// TIA Portal V20 export
FUNCTION "SafetyDoor" : Void   // FC97, LAD
// stored: SetENOAutomatically false
   VAR CONSTANT
      TRUE : Bool := TRUE;
      FALSE : Bool;
   END_VAR
   VAR_TEMP   // added for the SCL form of the ladder/FBD networks
      _w1 : Bool;
   END_VAR
BEGIN

REGION Network 1: fDoor1 monitoring
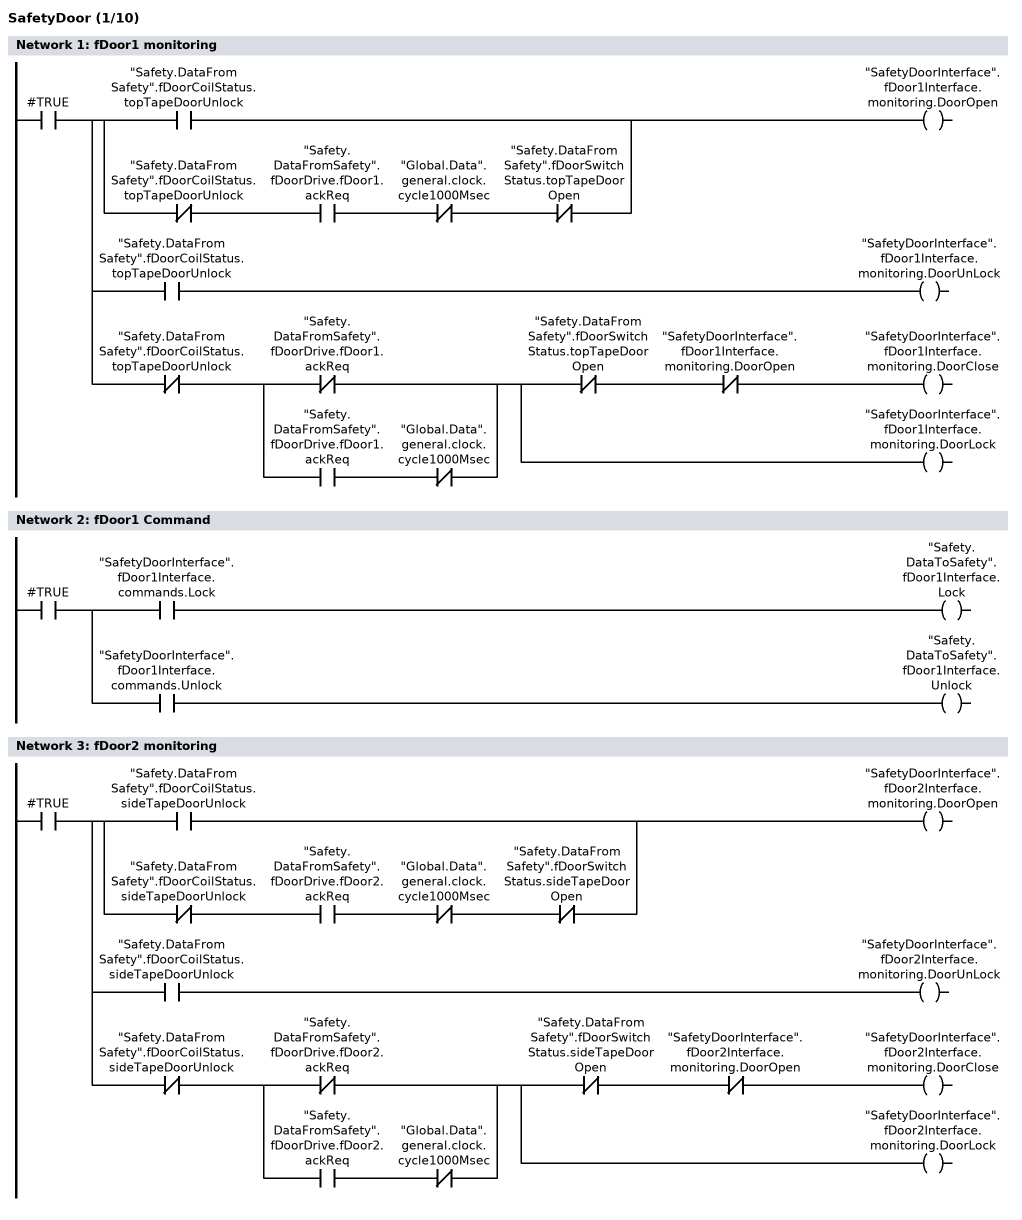
   RUNG wire#powerrail
      Contact( #TRUE )
      wire#w1
      Contact( "Safety.DataFromSafety".fDoorCoilStatus.topTapeDoorUnlock )
      wire#w2
      Coil( "SafetyDoorInterface".fDoor1Interface.monitoring.DoorOpen )
   END_RUNG
   RUNG wire#w1
      I_Contact( "Safety.DataFromSafety".fDoorCoilStatus.topTapeDoorUnlock )
      Contact( "Safety.DataFromSafety".fDoorDrive.fDoor1.ackReq )
      I_Contact( "Global.Data".general.clock.cycle1000Msec )
      I_Contact( "Safety.DataFromSafety".fDoorSwitchStatus.topTapeDoorOpen )
   END_RUNG wire#w2
   RUNG wire#w1
      Contact( "Safety.DataFromSafety".fDoorCoilStatus.topTapeDoorUnlock )
      Coil( "SafetyDoorInterface".fDoor1Interface.monitoring.DoorUnLock )
   END_RUNG
   RUNG wire#w1
      I_Contact( "Safety.DataFromSafety".fDoorCoilStatus.topTapeDoorUnlock )
      wire#w3
      I_Contact( "Safety.DataFromSafety".fDoorDrive.fDoor1.ackReq )
      wire#w4
      I_Contact( "Safety.DataFromSafety".fDoorSwitchStatus.topTapeDoorOpen )
      I_Contact( "SafetyDoorInterface".fDoor1Interface.monitoring.DoorOpen )
      Coil( "SafetyDoorInterface".fDoor1Interface.monitoring.DoorClose )
   END_RUNG
   RUNG wire#w3
      Contact( "Safety.DataFromSafety".fDoorDrive.fDoor1.ackReq )
      I_Contact( "Global.Data".general.clock.cycle1000Msec )
   END_RUNG wire#w4
   RUNG wire#w4
      Coil( "SafetyDoorInterface".fDoor1Interface.monitoring.DoorLock )
   END_RUNG
   // the same network as SCL:
   "SafetyDoorInterface".fDoor1Interface.monitoring.DoorOpen := #TRUE AND ("Safety.DataFromSafety".fDoorCoilStatus.topTapeDoorUnlock OR (NOT "Safety.DataFromSafety".fDoorCoilStatus.topTapeDoorUnlock AND "Safety.DataFromSafety".fDoorDrive.fDoor1.ackReq AND NOT "Global.Data".general.clock.cycle1000Msec AND NOT "Safety.DataFromSafety".fDoorSwitchStatus.topTapeDoorOpen));
   "SafetyDoorInterface".fDoor1Interface.monitoring.DoorUnLock := #TRUE AND "Safety.DataFromSafety".fDoorCoilStatus.topTapeDoorUnlock;
   #_w1 := #TRUE AND NOT "Safety.DataFromSafety".fDoorCoilStatus.topTapeDoorUnlock AND (NOT "Safety.DataFromSafety".fDoorDrive.fDoor1.ackReq OR ("Safety.DataFromSafety".fDoorDrive.fDoor1.ackReq AND NOT "Global.Data".general.clock.cycle1000Msec));
   "SafetyDoorInterface".fDoor1Interface.monitoring.DoorClose := #_w1 AND NOT "Safety.DataFromSafety".fDoorSwitchStatus.topTapeDoorOpen AND NOT "SafetyDoorInterface".fDoor1Interface.monitoring.DoorOpen;
   "SafetyDoorInterface".fDoor1Interface.monitoring.DoorLock := #_w1;
END_REGION

REGION Network 2: fDoor1 Command
   RUNG wire#powerrail
      Contact( #TRUE )
      wire#w1
      Contact( "SafetyDoorInterface".fDoor1Interface.commands.Lock )
      Coil( "Safety.DataToSafety".fDoor1Interface.Lock )
   END_RUNG
   RUNG wire#w1
      Contact( "SafetyDoorInterface".fDoor1Interface.commands.Unlock )
      Coil( "Safety.DataToSafety".fDoor1Interface.Unlock )
   END_RUNG
   // the same network as SCL:
   "Safety.DataToSafety".fDoor1Interface.Lock := #TRUE AND "SafetyDoorInterface".fDoor1Interface.commands.Lock;
   "Safety.DataToSafety".fDoor1Interface.Unlock := #TRUE AND "SafetyDoorInterface".fDoor1Interface.commands.Unlock;
END_REGION

REGION Network 3: fDoor2 monitoring
   RUNG wire#powerrail
      Contact( #TRUE )
      wire#w1
      Contact( "Safety.DataFromSafety".fDoorCoilStatus.sideTapeDoorUnlock )
      wire#w2
      Coil( "SafetyDoorInterface".fDoor2Interface.monitoring.DoorOpen )
   END_RUNG
   RUNG wire#w1
      I_Contact( "Safety.DataFromSafety".fDoorCoilStatus.sideTapeDoorUnlock )
      Contact( "Safety.DataFromSafety".fDoorDrive.fDoor2.ackReq )
      I_Contact( "Global.Data".general.clock.cycle1000Msec )
      I_Contact( "Safety.DataFromSafety".fDoorSwitchStatus.sideTapeDoorOpen )
   END_RUNG wire#w2
   RUNG wire#w1
      Contact( "Safety.DataFromSafety".fDoorCoilStatus.sideTapeDoorUnlock )
      Coil( "SafetyDoorInterface".fDoor2Interface.monitoring.DoorUnLock )
   END_RUNG
   RUNG wire#w1
      I_Contact( "Safety.DataFromSafety".fDoorCoilStatus.sideTapeDoorUnlock )
      wire#w3
      I_Contact( "Safety.DataFromSafety".fDoorDrive.fDoor2.ackReq )
      wire#w4
      I_Contact( "Safety.DataFromSafety".fDoorSwitchStatus.sideTapeDoorOpen )
      I_Contact( "SafetyDoorInterface".fDoor2Interface.monitoring.DoorOpen )
      Coil( "SafetyDoorInterface".fDoor2Interface.monitoring.DoorClose )
   END_RUNG
   RUNG wire#w3
      Contact( "Safety.DataFromSafety".fDoorDrive.fDoor2.ackReq )
      I_Contact( "Global.Data".general.clock.cycle1000Msec )
   END_RUNG wire#w4
   RUNG wire#w4
      Coil( "SafetyDoorInterface".fDoor2Interface.monitoring.DoorLock )
   END_RUNG
   // the same network as SCL:
   "SafetyDoorInterface".fDoor2Interface.monitoring.DoorOpen := #TRUE AND ("Safety.DataFromSafety".fDoorCoilStatus.sideTapeDoorUnlock OR (NOT "Safety.DataFromSafety".fDoorCoilStatus.sideTapeDoorUnlock AND "Safety.DataFromSafety".fDoorDrive.fDoor2.ackReq AND NOT "Global.Data".general.clock.cycle1000Msec AND NOT "Safety.DataFromSafety".fDoorSwitchStatus.sideTapeDoorOpen));
   "SafetyDoorInterface".fDoor2Interface.monitoring.DoorUnLock := #TRUE AND "Safety.DataFromSafety".fDoorCoilStatus.sideTapeDoorUnlock;
   #_w1 := #TRUE AND NOT "Safety.DataFromSafety".fDoorCoilStatus.sideTapeDoorUnlock AND (NOT "Safety.DataFromSafety".fDoorDrive.fDoor2.ackReq OR ("Safety.DataFromSafety".fDoorDrive.fDoor2.ackReq AND NOT "Global.Data".general.clock.cycle1000Msec));
   "SafetyDoorInterface".fDoor2Interface.monitoring.DoorClose := #_w1 AND NOT "Safety.DataFromSafety".fDoorSwitchStatus.sideTapeDoorOpen AND NOT "SafetyDoorInterface".fDoor2Interface.monitoring.DoorOpen;
   "SafetyDoorInterface".fDoor2Interface.monitoring.DoorLock := #_w1;
END_REGION

REGION Network 4: fDoor2 Command
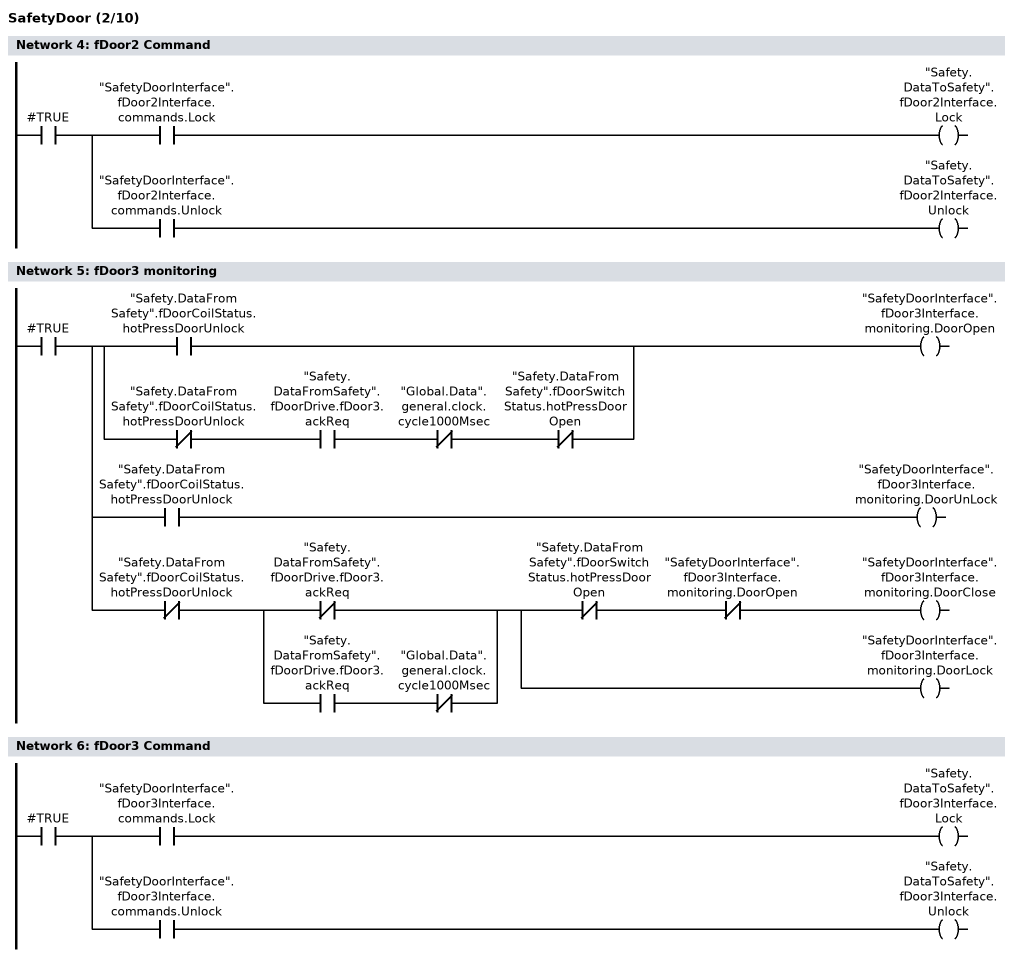
   RUNG wire#powerrail
      Contact( #TRUE )
      wire#w1
      Contact( "SafetyDoorInterface".fDoor2Interface.commands.Lock )
      Coil( "Safety.DataToSafety".fDoor2Interface.Lock )
   END_RUNG
   RUNG wire#w1
      Contact( "SafetyDoorInterface".fDoor2Interface.commands.Unlock )
      Coil( "Safety.DataToSafety".fDoor2Interface.Unlock )
   END_RUNG
   // the same network as SCL:
   "Safety.DataToSafety".fDoor2Interface.Lock := #TRUE AND "SafetyDoorInterface".fDoor2Interface.commands.Lock;
   "Safety.DataToSafety".fDoor2Interface.Unlock := #TRUE AND "SafetyDoorInterface".fDoor2Interface.commands.Unlock;
END_REGION

REGION Network 5: fDoor3 monitoring
   RUNG wire#powerrail
      Contact( #TRUE )
      wire#w1
      Contact( "Safety.DataFromSafety".fDoorCoilStatus.hotPressDoorUnlock )
      wire#w2
      Coil( "SafetyDoorInterface".fDoor3Interface.monitoring.DoorOpen )
   END_RUNG
   RUNG wire#w1
      I_Contact( "Safety.DataFromSafety".fDoorCoilStatus.hotPressDoorUnlock )
      Contact( "Safety.DataFromSafety".fDoorDrive.fDoor3.ackReq )
      I_Contact( "Global.Data".general.clock.cycle1000Msec )
      I_Contact( "Safety.DataFromSafety".fDoorSwitchStatus.hotPressDoorOpen )
   END_RUNG wire#w2
   RUNG wire#w1
      Contact( "Safety.DataFromSafety".fDoorCoilStatus.hotPressDoorUnlock )
      Coil( "SafetyDoorInterface".fDoor3Interface.monitoring.DoorUnLock )
   END_RUNG
   RUNG wire#w1
      I_Contact( "Safety.DataFromSafety".fDoorCoilStatus.hotPressDoorUnlock )
      wire#w3
      I_Contact( "Safety.DataFromSafety".fDoorDrive.fDoor3.ackReq )
      wire#w4
      I_Contact( "Safety.DataFromSafety".fDoorSwitchStatus.hotPressDoorOpen )
      I_Contact( "SafetyDoorInterface".fDoor3Interface.monitoring.DoorOpen )
      Coil( "SafetyDoorInterface".fDoor3Interface.monitoring.DoorClose )
   END_RUNG
   RUNG wire#w3
      Contact( "Safety.DataFromSafety".fDoorDrive.fDoor3.ackReq )
      I_Contact( "Global.Data".general.clock.cycle1000Msec )
   END_RUNG wire#w4
   RUNG wire#w4
      Coil( "SafetyDoorInterface".fDoor3Interface.monitoring.DoorLock )
   END_RUNG
   // the same network as SCL:
   "SafetyDoorInterface".fDoor3Interface.monitoring.DoorOpen := #TRUE AND ("Safety.DataFromSafety".fDoorCoilStatus.hotPressDoorUnlock OR (NOT "Safety.DataFromSafety".fDoorCoilStatus.hotPressDoorUnlock AND "Safety.DataFromSafety".fDoorDrive.fDoor3.ackReq AND NOT "Global.Data".general.clock.cycle1000Msec AND NOT "Safety.DataFromSafety".fDoorSwitchStatus.hotPressDoorOpen));
   "SafetyDoorInterface".fDoor3Interface.monitoring.DoorUnLock := #TRUE AND "Safety.DataFromSafety".fDoorCoilStatus.hotPressDoorUnlock;
   #_w1 := #TRUE AND NOT "Safety.DataFromSafety".fDoorCoilStatus.hotPressDoorUnlock AND (NOT "Safety.DataFromSafety".fDoorDrive.fDoor3.ackReq OR ("Safety.DataFromSafety".fDoorDrive.fDoor3.ackReq AND NOT "Global.Data".general.clock.cycle1000Msec));
   "SafetyDoorInterface".fDoor3Interface.monitoring.DoorClose := #_w1 AND NOT "Safety.DataFromSafety".fDoorSwitchStatus.hotPressDoorOpen AND NOT "SafetyDoorInterface".fDoor3Interface.monitoring.DoorOpen;
   "SafetyDoorInterface".fDoor3Interface.monitoring.DoorLock := #_w1;
END_REGION

REGION Network 6: fDoor3 Command
   RUNG wire#powerrail
      Contact( #TRUE )
      wire#w1
      Contact( "SafetyDoorInterface".fDoor3Interface.commands.Lock )
      Coil( "Safety.DataToSafety".fDoor3Interface.Lock )
   END_RUNG
   RUNG wire#w1
      Contact( "SafetyDoorInterface".fDoor3Interface.commands.Unlock )
      Coil( "Safety.DataToSafety".fDoor3Interface.Unlock )
   END_RUNG
   // the same network as SCL:
   "Safety.DataToSafety".fDoor3Interface.Lock := #TRUE AND "SafetyDoorInterface".fDoor3Interface.commands.Lock;
   "Safety.DataToSafety".fDoor3Interface.Unlock := #TRUE AND "SafetyDoorInterface".fDoor3Interface.commands.Unlock;
END_REGION

REGION Network 7: fDoor4 monitoring
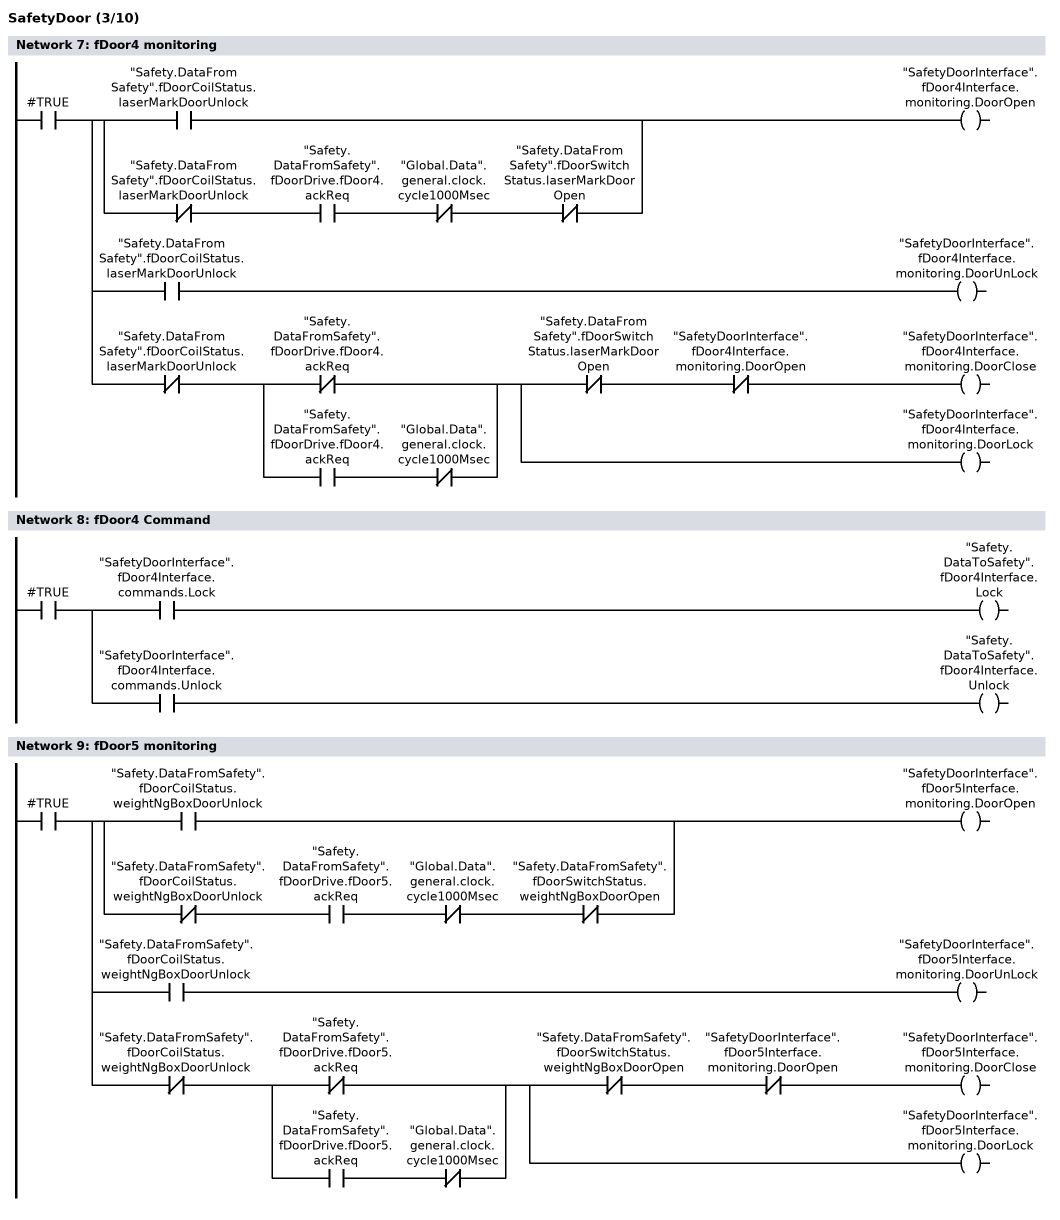
   RUNG wire#powerrail
      Contact( #TRUE )
      wire#w1
      Contact( "Safety.DataFromSafety".fDoorCoilStatus.laserMarkDoorUnlock )
      wire#w2
      Coil( "SafetyDoorInterface".fDoor4Interface.monitoring.DoorOpen )
   END_RUNG
   RUNG wire#w1
      I_Contact( "Safety.DataFromSafety".fDoorCoilStatus.laserMarkDoorUnlock )
      Contact( "Safety.DataFromSafety".fDoorDrive.fDoor4.ackReq )
      I_Contact( "Global.Data".general.clock.cycle1000Msec )
      I_Contact( "Safety.DataFromSafety".fDoorSwitchStatus.laserMarkDoorOpen )
   END_RUNG wire#w2
   RUNG wire#w1
      Contact( "Safety.DataFromSafety".fDoorCoilStatus.laserMarkDoorUnlock )
      Coil( "SafetyDoorInterface".fDoor4Interface.monitoring.DoorUnLock )
   END_RUNG
   RUNG wire#w1
      I_Contact( "Safety.DataFromSafety".fDoorCoilStatus.laserMarkDoorUnlock )
      wire#w3
      I_Contact( "Safety.DataFromSafety".fDoorDrive.fDoor4.ackReq )
      wire#w4
      I_Contact( "Safety.DataFromSafety".fDoorSwitchStatus.laserMarkDoorOpen )
      I_Contact( "SafetyDoorInterface".fDoor4Interface.monitoring.DoorOpen )
      Coil( "SafetyDoorInterface".fDoor4Interface.monitoring.DoorClose )
   END_RUNG
   RUNG wire#w3
      Contact( "Safety.DataFromSafety".fDoorDrive.fDoor4.ackReq )
      I_Contact( "Global.Data".general.clock.cycle1000Msec )
   END_RUNG wire#w4
   RUNG wire#w4
      Coil( "SafetyDoorInterface".fDoor4Interface.monitoring.DoorLock )
   END_RUNG
   // the same network as SCL:
   "SafetyDoorInterface".fDoor4Interface.monitoring.DoorOpen := #TRUE AND ("Safety.DataFromSafety".fDoorCoilStatus.laserMarkDoorUnlock OR (NOT "Safety.DataFromSafety".fDoorCoilStatus.laserMarkDoorUnlock AND "Safety.DataFromSafety".fDoorDrive.fDoor4.ackReq AND NOT "Global.Data".general.clock.cycle1000Msec AND NOT "Safety.DataFromSafety".fDoorSwitchStatus.laserMarkDoorOpen));
   "SafetyDoorInterface".fDoor4Interface.monitoring.DoorUnLock := #TRUE AND "Safety.DataFromSafety".fDoorCoilStatus.laserMarkDoorUnlock;
   #_w1 := #TRUE AND NOT "Safety.DataFromSafety".fDoorCoilStatus.laserMarkDoorUnlock AND (NOT "Safety.DataFromSafety".fDoorDrive.fDoor4.ackReq OR ("Safety.DataFromSafety".fDoorDrive.fDoor4.ackReq AND NOT "Global.Data".general.clock.cycle1000Msec));
   "SafetyDoorInterface".fDoor4Interface.monitoring.DoorClose := #_w1 AND NOT "Safety.DataFromSafety".fDoorSwitchStatus.laserMarkDoorOpen AND NOT "SafetyDoorInterface".fDoor4Interface.monitoring.DoorOpen;
   "SafetyDoorInterface".fDoor4Interface.monitoring.DoorLock := #_w1;
END_REGION

REGION Network 8: fDoor4 Command
   RUNG wire#powerrail
      Contact( #TRUE )
      wire#w1
      Contact( "SafetyDoorInterface".fDoor4Interface.commands.Lock )
      Coil( "Safety.DataToSafety".fDoor4Interface.Lock )
   END_RUNG
   RUNG wire#w1
      Contact( "SafetyDoorInterface".fDoor4Interface.commands.Unlock )
      Coil( "Safety.DataToSafety".fDoor4Interface.Unlock )
   END_RUNG
   // the same network as SCL:
   "Safety.DataToSafety".fDoor4Interface.Lock := #TRUE AND "SafetyDoorInterface".fDoor4Interface.commands.Lock;
   "Safety.DataToSafety".fDoor4Interface.Unlock := #TRUE AND "SafetyDoorInterface".fDoor4Interface.commands.Unlock;
END_REGION

REGION Network 9: fDoor5 monitoring
   RUNG wire#powerrail
      Contact( #TRUE )
      wire#w1
      Contact( "Safety.DataFromSafety".fDoorCoilStatus.weightNgBoxDoorUnlock )
      wire#w2
      Coil( "SafetyDoorInterface".fDoor5Interface.monitoring.DoorOpen )
   END_RUNG
   RUNG wire#w1
      I_Contact( "Safety.DataFromSafety".fDoorCoilStatus.weightNgBoxDoorUnlock )
      Contact( "Safety.DataFromSafety".fDoorDrive.fDoor5.ackReq )
      I_Contact( "Global.Data".general.clock.cycle1000Msec )
      I_Contact( "Safety.DataFromSafety".fDoorSwitchStatus.weightNgBoxDoorOpen )
   END_RUNG wire#w2
   RUNG wire#w1
      Contact( "Safety.DataFromSafety".fDoorCoilStatus.weightNgBoxDoorUnlock )
      Coil( "SafetyDoorInterface".fDoor5Interface.monitoring.DoorUnLock )
   END_RUNG
   RUNG wire#w1
      I_Contact( "Safety.DataFromSafety".fDoorCoilStatus.weightNgBoxDoorUnlock )
      wire#w3
      I_Contact( "Safety.DataFromSafety".fDoorDrive.fDoor5.ackReq )
      wire#w4
      I_Contact( "Safety.DataFromSafety".fDoorSwitchStatus.weightNgBoxDoorOpen )
      I_Contact( "SafetyDoorInterface".fDoor5Interface.monitoring.DoorOpen )
      Coil( "SafetyDoorInterface".fDoor5Interface.monitoring.DoorClose )
   END_RUNG
   RUNG wire#w3
      Contact( "Safety.DataFromSafety".fDoorDrive.fDoor5.ackReq )
      I_Contact( "Global.Data".general.clock.cycle1000Msec )
   END_RUNG wire#w4
   RUNG wire#w4
      Coil( "SafetyDoorInterface".fDoor5Interface.monitoring.DoorLock )
   END_RUNG
   // the same network as SCL:
   "SafetyDoorInterface".fDoor5Interface.monitoring.DoorOpen := #TRUE AND ("Safety.DataFromSafety".fDoorCoilStatus.weightNgBoxDoorUnlock OR (NOT "Safety.DataFromSafety".fDoorCoilStatus.weightNgBoxDoorUnlock AND "Safety.DataFromSafety".fDoorDrive.fDoor5.ackReq AND NOT "Global.Data".general.clock.cycle1000Msec AND NOT "Safety.DataFromSafety".fDoorSwitchStatus.weightNgBoxDoorOpen));
   "SafetyDoorInterface".fDoor5Interface.monitoring.DoorUnLock := #TRUE AND "Safety.DataFromSafety".fDoorCoilStatus.weightNgBoxDoorUnlock;
   #_w1 := #TRUE AND NOT "Safety.DataFromSafety".fDoorCoilStatus.weightNgBoxDoorUnlock AND (NOT "Safety.DataFromSafety".fDoorDrive.fDoor5.ackReq OR ("Safety.DataFromSafety".fDoorDrive.fDoor5.ackReq AND NOT "Global.Data".general.clock.cycle1000Msec));
   "SafetyDoorInterface".fDoor5Interface.monitoring.DoorClose := #_w1 AND NOT "Safety.DataFromSafety".fDoorSwitchStatus.weightNgBoxDoorOpen AND NOT "SafetyDoorInterface".fDoor5Interface.monitoring.DoorOpen;
   "SafetyDoorInterface".fDoor5Interface.monitoring.DoorLock := #_w1;
END_REGION

REGION Network 10: fDoor5 Command
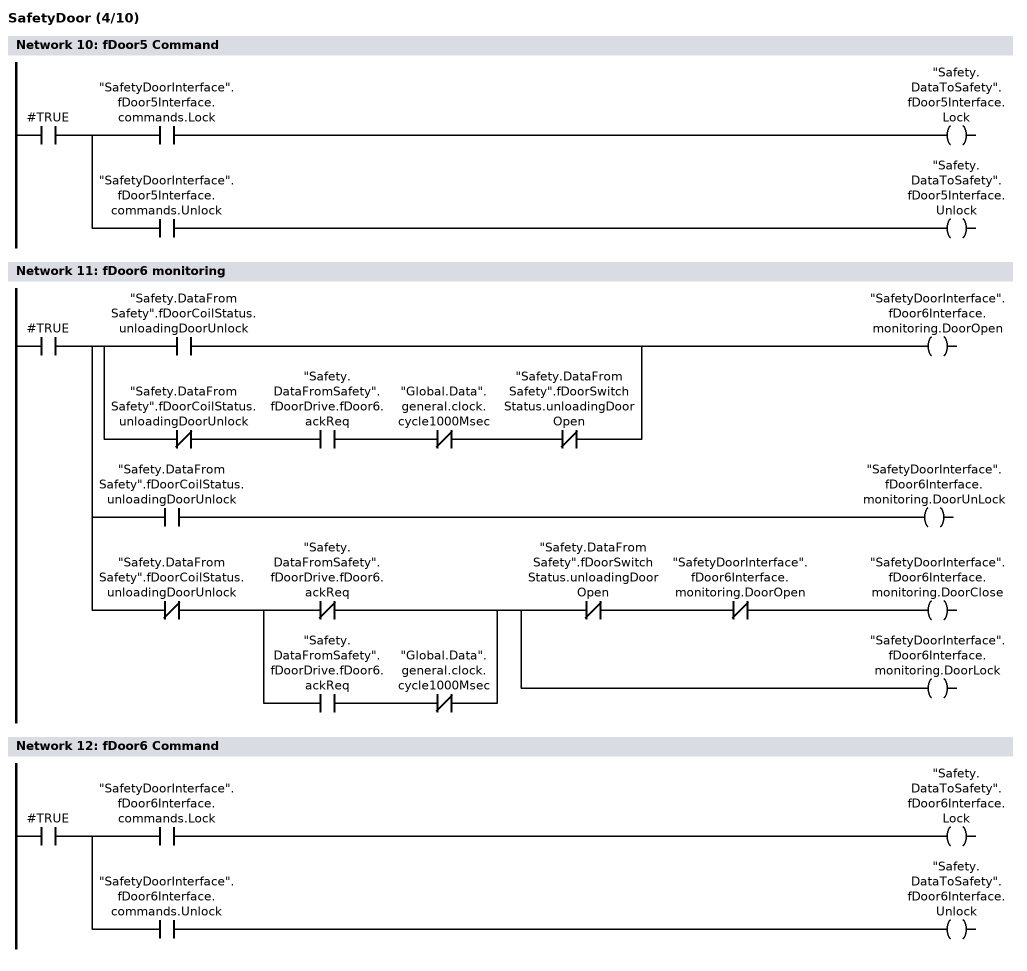
   RUNG wire#powerrail
      Contact( #TRUE )
      wire#w1
      Contact( "SafetyDoorInterface".fDoor5Interface.commands.Lock )
      Coil( "Safety.DataToSafety".fDoor5Interface.Lock )
   END_RUNG
   RUNG wire#w1
      Contact( "SafetyDoorInterface".fDoor5Interface.commands.Unlock )
      Coil( "Safety.DataToSafety".fDoor5Interface.Unlock )
   END_RUNG
   // the same network as SCL:
   "Safety.DataToSafety".fDoor5Interface.Lock := #TRUE AND "SafetyDoorInterface".fDoor5Interface.commands.Lock;
   "Safety.DataToSafety".fDoor5Interface.Unlock := #TRUE AND "SafetyDoorInterface".fDoor5Interface.commands.Unlock;
END_REGION

REGION Network 11: fDoor6 monitoring
   RUNG wire#powerrail
      Contact( #TRUE )
      wire#w1
      Contact( "Safety.DataFromSafety".fDoorCoilStatus.unloadingDoorUnlock )
      wire#w2
      Coil( "SafetyDoorInterface".fDoor6Interface.monitoring.DoorOpen )
   END_RUNG
   RUNG wire#w1
      I_Contact( "Safety.DataFromSafety".fDoorCoilStatus.unloadingDoorUnlock )
      Contact( "Safety.DataFromSafety".fDoorDrive.fDoor6.ackReq )
      I_Contact( "Global.Data".general.clock.cycle1000Msec )
      I_Contact( "Safety.DataFromSafety".fDoorSwitchStatus.unloadingDoorOpen )
   END_RUNG wire#w2
   RUNG wire#w1
      Contact( "Safety.DataFromSafety".fDoorCoilStatus.unloadingDoorUnlock )
      Coil( "SafetyDoorInterface".fDoor6Interface.monitoring.DoorUnLock )
   END_RUNG
   RUNG wire#w1
      I_Contact( "Safety.DataFromSafety".fDoorCoilStatus.unloadingDoorUnlock )
      wire#w3
      I_Contact( "Safety.DataFromSafety".fDoorDrive.fDoor6.ackReq )
      wire#w4
      I_Contact( "Safety.DataFromSafety".fDoorSwitchStatus.unloadingDoorOpen )
      I_Contact( "SafetyDoorInterface".fDoor6Interface.monitoring.DoorOpen )
      Coil( "SafetyDoorInterface".fDoor6Interface.monitoring.DoorClose )
   END_RUNG
   RUNG wire#w3
      Contact( "Safety.DataFromSafety".fDoorDrive.fDoor6.ackReq )
      I_Contact( "Global.Data".general.clock.cycle1000Msec )
   END_RUNG wire#w4
   RUNG wire#w4
      Coil( "SafetyDoorInterface".fDoor6Interface.monitoring.DoorLock )
   END_RUNG
   // the same network as SCL:
   "SafetyDoorInterface".fDoor6Interface.monitoring.DoorOpen := #TRUE AND ("Safety.DataFromSafety".fDoorCoilStatus.unloadingDoorUnlock OR (NOT "Safety.DataFromSafety".fDoorCoilStatus.unloadingDoorUnlock AND "Safety.DataFromSafety".fDoorDrive.fDoor6.ackReq AND NOT "Global.Data".general.clock.cycle1000Msec AND NOT "Safety.DataFromSafety".fDoorSwitchStatus.unloadingDoorOpen));
   "SafetyDoorInterface".fDoor6Interface.monitoring.DoorUnLock := #TRUE AND "Safety.DataFromSafety".fDoorCoilStatus.unloadingDoorUnlock;
   #_w1 := #TRUE AND NOT "Safety.DataFromSafety".fDoorCoilStatus.unloadingDoorUnlock AND (NOT "Safety.DataFromSafety".fDoorDrive.fDoor6.ackReq OR ("Safety.DataFromSafety".fDoorDrive.fDoor6.ackReq AND NOT "Global.Data".general.clock.cycle1000Msec));
   "SafetyDoorInterface".fDoor6Interface.monitoring.DoorClose := #_w1 AND NOT "Safety.DataFromSafety".fDoorSwitchStatus.unloadingDoorOpen AND NOT "SafetyDoorInterface".fDoor6Interface.monitoring.DoorOpen;
   "SafetyDoorInterface".fDoor6Interface.monitoring.DoorLock := #_w1;
END_REGION

REGION Network 12: fDoor6 Command
   RUNG wire#powerrail
      Contact( #TRUE )
      wire#w1
      Contact( "SafetyDoorInterface".fDoor6Interface.commands.Lock )
      Coil( "Safety.DataToSafety".fDoor6Interface.Lock )
   END_RUNG
   RUNG wire#w1
      Contact( "SafetyDoorInterface".fDoor6Interface.commands.Unlock )
      Coil( "Safety.DataToSafety".fDoor6Interface.Unlock )
   END_RUNG
   // the same network as SCL:
   "Safety.DataToSafety".fDoor6Interface.Lock := #TRUE AND "SafetyDoorInterface".fDoor6Interface.commands.Lock;
   "Safety.DataToSafety".fDoor6Interface.Unlock := #TRUE AND "SafetyDoorInterface".fDoor6Interface.commands.Unlock;
END_REGION

REGION Network 13: fDoor7 monitoring
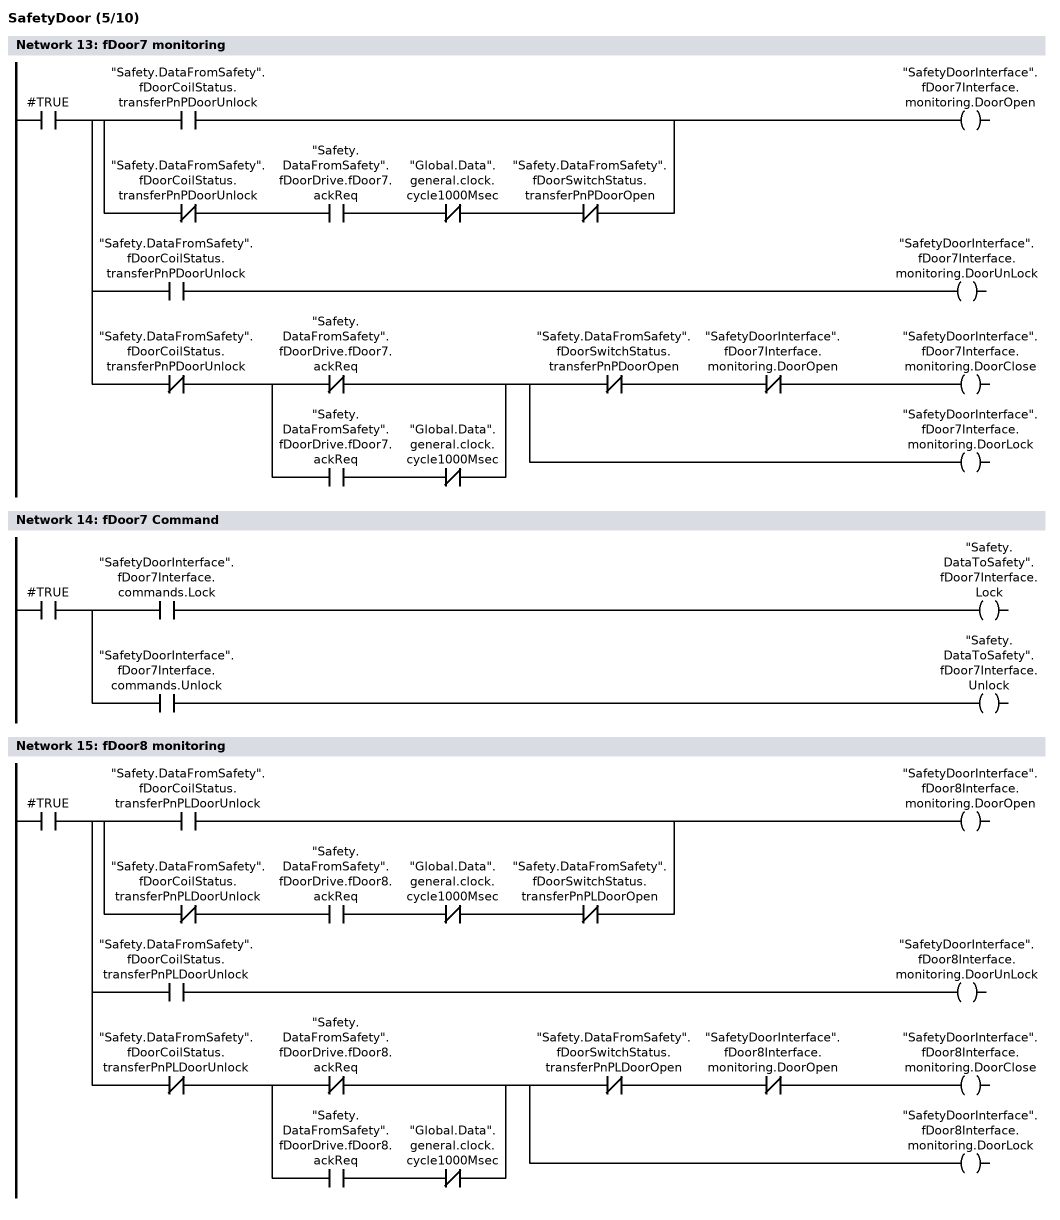
   RUNG wire#powerrail
      Contact( #TRUE )
      wire#w1
      Contact( "Safety.DataFromSafety".fDoorCoilStatus.transferPnPDoorUnlock )
      wire#w2
      Coil( "SafetyDoorInterface".fDoor7Interface.monitoring.DoorOpen )
   END_RUNG
   RUNG wire#w1
      I_Contact( "Safety.DataFromSafety".fDoorCoilStatus.transferPnPDoorUnlock )
      Contact( "Safety.DataFromSafety".fDoorDrive.fDoor7.ackReq )
      I_Contact( "Global.Data".general.clock.cycle1000Msec )
      I_Contact( "Safety.DataFromSafety".fDoorSwitchStatus.transferPnPDoorOpen )
   END_RUNG wire#w2
   RUNG wire#w1
      Contact( "Safety.DataFromSafety".fDoorCoilStatus.transferPnPDoorUnlock )
      Coil( "SafetyDoorInterface".fDoor7Interface.monitoring.DoorUnLock )
   END_RUNG
   RUNG wire#w1
      I_Contact( "Safety.DataFromSafety".fDoorCoilStatus.transferPnPDoorUnlock )
      wire#w3
      I_Contact( "Safety.DataFromSafety".fDoorDrive.fDoor7.ackReq )
      wire#w4
      I_Contact( "Safety.DataFromSafety".fDoorSwitchStatus.transferPnPDoorOpen )
      I_Contact( "SafetyDoorInterface".fDoor7Interface.monitoring.DoorOpen )
      Coil( "SafetyDoorInterface".fDoor7Interface.monitoring.DoorClose )
   END_RUNG
   RUNG wire#w3
      Contact( "Safety.DataFromSafety".fDoorDrive.fDoor7.ackReq )
      I_Contact( "Global.Data".general.clock.cycle1000Msec )
   END_RUNG wire#w4
   RUNG wire#w4
      Coil( "SafetyDoorInterface".fDoor7Interface.monitoring.DoorLock )
   END_RUNG
   // the same network as SCL:
   "SafetyDoorInterface".fDoor7Interface.monitoring.DoorOpen := #TRUE AND ("Safety.DataFromSafety".fDoorCoilStatus.transferPnPDoorUnlock OR (NOT "Safety.DataFromSafety".fDoorCoilStatus.transferPnPDoorUnlock AND "Safety.DataFromSafety".fDoorDrive.fDoor7.ackReq AND NOT "Global.Data".general.clock.cycle1000Msec AND NOT "Safety.DataFromSafety".fDoorSwitchStatus.transferPnPDoorOpen));
   "SafetyDoorInterface".fDoor7Interface.monitoring.DoorUnLock := #TRUE AND "Safety.DataFromSafety".fDoorCoilStatus.transferPnPDoorUnlock;
   #_w1 := #TRUE AND NOT "Safety.DataFromSafety".fDoorCoilStatus.transferPnPDoorUnlock AND (NOT "Safety.DataFromSafety".fDoorDrive.fDoor7.ackReq OR ("Safety.DataFromSafety".fDoorDrive.fDoor7.ackReq AND NOT "Global.Data".general.clock.cycle1000Msec));
   "SafetyDoorInterface".fDoor7Interface.monitoring.DoorClose := #_w1 AND NOT "Safety.DataFromSafety".fDoorSwitchStatus.transferPnPDoorOpen AND NOT "SafetyDoorInterface".fDoor7Interface.monitoring.DoorOpen;
   "SafetyDoorInterface".fDoor7Interface.monitoring.DoorLock := #_w1;
END_REGION

REGION Network 14: fDoor7 Command
   RUNG wire#powerrail
      Contact( #TRUE )
      wire#w1
      Contact( "SafetyDoorInterface".fDoor7Interface.commands.Lock )
      Coil( "Safety.DataToSafety".fDoor7Interface.Lock )
   END_RUNG
   RUNG wire#w1
      Contact( "SafetyDoorInterface".fDoor7Interface.commands.Unlock )
      Coil( "Safety.DataToSafety".fDoor7Interface.Unlock )
   END_RUNG
   // the same network as SCL:
   "Safety.DataToSafety".fDoor7Interface.Lock := #TRUE AND "SafetyDoorInterface".fDoor7Interface.commands.Lock;
   "Safety.DataToSafety".fDoor7Interface.Unlock := #TRUE AND "SafetyDoorInterface".fDoor7Interface.commands.Unlock;
END_REGION

REGION Network 15: fDoor8 monitoring
   RUNG wire#powerrail
      Contact( #TRUE )
      wire#w1
      Contact( "Safety.DataFromSafety".fDoorCoilStatus.transferPnPLDoorUnlock )
      wire#w2
      Coil( "SafetyDoorInterface".fDoor8Interface.monitoring.DoorOpen )
   END_RUNG
   RUNG wire#w1
      I_Contact( "Safety.DataFromSafety".fDoorCoilStatus.transferPnPLDoorUnlock )
      Contact( "Safety.DataFromSafety".fDoorDrive.fDoor8.ackReq )
      I_Contact( "Global.Data".general.clock.cycle1000Msec )
      I_Contact( "Safety.DataFromSafety".fDoorSwitchStatus.transferPnPLDoorOpen )
   END_RUNG wire#w2
   RUNG wire#w1
      Contact( "Safety.DataFromSafety".fDoorCoilStatus.transferPnPLDoorUnlock )
      Coil( "SafetyDoorInterface".fDoor8Interface.monitoring.DoorUnLock )
   END_RUNG
   RUNG wire#w1
      I_Contact( "Safety.DataFromSafety".fDoorCoilStatus.transferPnPLDoorUnlock )
      wire#w3
      I_Contact( "Safety.DataFromSafety".fDoorDrive.fDoor8.ackReq )
      wire#w4
      I_Contact( "Safety.DataFromSafety".fDoorSwitchStatus.transferPnPLDoorOpen )
      I_Contact( "SafetyDoorInterface".fDoor8Interface.monitoring.DoorOpen )
      Coil( "SafetyDoorInterface".fDoor8Interface.monitoring.DoorClose )
   END_RUNG
   RUNG wire#w3
      Contact( "Safety.DataFromSafety".fDoorDrive.fDoor8.ackReq )
      I_Contact( "Global.Data".general.clock.cycle1000Msec )
   END_RUNG wire#w4
   RUNG wire#w4
      Coil( "SafetyDoorInterface".fDoor8Interface.monitoring.DoorLock )
   END_RUNG
   // the same network as SCL:
   "SafetyDoorInterface".fDoor8Interface.monitoring.DoorOpen := #TRUE AND ("Safety.DataFromSafety".fDoorCoilStatus.transferPnPLDoorUnlock OR (NOT "Safety.DataFromSafety".fDoorCoilStatus.transferPnPLDoorUnlock AND "Safety.DataFromSafety".fDoorDrive.fDoor8.ackReq AND NOT "Global.Data".general.clock.cycle1000Msec AND NOT "Safety.DataFromSafety".fDoorSwitchStatus.transferPnPLDoorOpen));
   "SafetyDoorInterface".fDoor8Interface.monitoring.DoorUnLock := #TRUE AND "Safety.DataFromSafety".fDoorCoilStatus.transferPnPLDoorUnlock;
   #_w1 := #TRUE AND NOT "Safety.DataFromSafety".fDoorCoilStatus.transferPnPLDoorUnlock AND (NOT "Safety.DataFromSafety".fDoorDrive.fDoor8.ackReq OR ("Safety.DataFromSafety".fDoorDrive.fDoor8.ackReq AND NOT "Global.Data".general.clock.cycle1000Msec));
   "SafetyDoorInterface".fDoor8Interface.monitoring.DoorClose := #_w1 AND NOT "Safety.DataFromSafety".fDoorSwitchStatus.transferPnPLDoorOpen AND NOT "SafetyDoorInterface".fDoor8Interface.monitoring.DoorOpen;
   "SafetyDoorInterface".fDoor8Interface.monitoring.DoorLock := #_w1;
END_REGION

REGION Network 16: fDoor8 Command
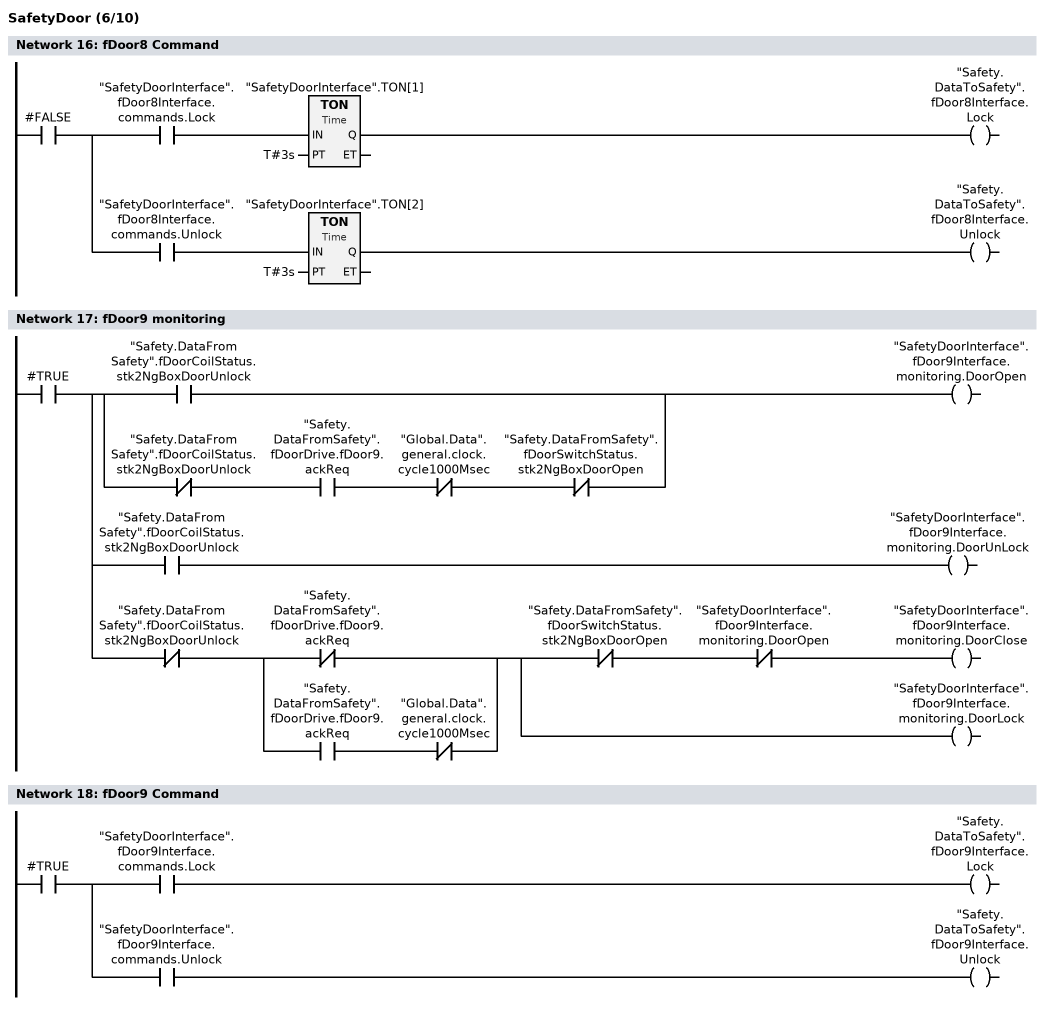
   RUNG wire#powerrail
      Contact( #FALSE )
      wire#w1
      Contact( "SafetyDoorInterface".fDoor8Interface.commands.Lock )
      { S7_Templates := "time_type := Time" } "SafetyDoorInterface".TON[1].TON(pt := T#3s, et =>)
      Coil( "Safety.DataToSafety".fDoor8Interface.Lock )
   END_RUNG
   RUNG wire#w1
      Contact( "SafetyDoorInterface".fDoor8Interface.commands.Unlock )
      { S7_Templates := "time_type := Time" } "SafetyDoorInterface".TON[2].TON(pt := T#3s, et =>)
      Coil( "Safety.DataToSafety".fDoor8Interface.Unlock )
   END_RUNG
   // the same network as SCL:
   "SafetyDoorInterface".TON[1].TON(IN := #FALSE AND "SafetyDoorInterface".fDoor8Interface.commands.Lock,
                           PT := T#3s);
   "Safety.DataToSafety".fDoor8Interface.Lock := "SafetyDoorInterface".TON[1].Q;
   "SafetyDoorInterface".TON[2].TON(IN := #FALSE AND "SafetyDoorInterface".fDoor8Interface.commands.Unlock,
                           PT := T#3s);
   "Safety.DataToSafety".fDoor8Interface.Unlock := "SafetyDoorInterface".TON[2].Q;
END_REGION

REGION Network 17: fDoor9 monitoring
   RUNG wire#powerrail
      Contact( #TRUE )
      wire#w1
      Contact( "Safety.DataFromSafety".fDoorCoilStatus.stk2NgBoxDoorUnlock )
      wire#w2
      Coil( "SafetyDoorInterface".fDoor9Interface.monitoring.DoorOpen )
   END_RUNG
   RUNG wire#w1
      I_Contact( "Safety.DataFromSafety".fDoorCoilStatus.stk2NgBoxDoorUnlock )
      Contact( "Safety.DataFromSafety".fDoorDrive.fDoor9.ackReq )
      I_Contact( "Global.Data".general.clock.cycle1000Msec )
      I_Contact( "Safety.DataFromSafety".fDoorSwitchStatus.stk2NgBoxDoorOpen )
   END_RUNG wire#w2
   RUNG wire#w1
      Contact( "Safety.DataFromSafety".fDoorCoilStatus.stk2NgBoxDoorUnlock )
      Coil( "SafetyDoorInterface".fDoor9Interface.monitoring.DoorUnLock )
   END_RUNG
   RUNG wire#w1
      I_Contact( "Safety.DataFromSafety".fDoorCoilStatus.stk2NgBoxDoorUnlock )
      wire#w3
      I_Contact( "Safety.DataFromSafety".fDoorDrive.fDoor9.ackReq )
      wire#w4
      I_Contact( "Safety.DataFromSafety".fDoorSwitchStatus.stk2NgBoxDoorOpen )
      I_Contact( "SafetyDoorInterface".fDoor9Interface.monitoring.DoorOpen )
      Coil( "SafetyDoorInterface".fDoor9Interface.monitoring.DoorClose )
   END_RUNG
   RUNG wire#w3
      Contact( "Safety.DataFromSafety".fDoorDrive.fDoor9.ackReq )
      I_Contact( "Global.Data".general.clock.cycle1000Msec )
   END_RUNG wire#w4
   RUNG wire#w4
      Coil( "SafetyDoorInterface".fDoor9Interface.monitoring.DoorLock )
   END_RUNG
   // the same network as SCL:
   "SafetyDoorInterface".fDoor9Interface.monitoring.DoorOpen := #TRUE AND ("Safety.DataFromSafety".fDoorCoilStatus.stk2NgBoxDoorUnlock OR (NOT "Safety.DataFromSafety".fDoorCoilStatus.stk2NgBoxDoorUnlock AND "Safety.DataFromSafety".fDoorDrive.fDoor9.ackReq AND NOT "Global.Data".general.clock.cycle1000Msec AND NOT "Safety.DataFromSafety".fDoorSwitchStatus.stk2NgBoxDoorOpen));
   "SafetyDoorInterface".fDoor9Interface.monitoring.DoorUnLock := #TRUE AND "Safety.DataFromSafety".fDoorCoilStatus.stk2NgBoxDoorUnlock;
   #_w1 := #TRUE AND NOT "Safety.DataFromSafety".fDoorCoilStatus.stk2NgBoxDoorUnlock AND (NOT "Safety.DataFromSafety".fDoorDrive.fDoor9.ackReq OR ("Safety.DataFromSafety".fDoorDrive.fDoor9.ackReq AND NOT "Global.Data".general.clock.cycle1000Msec));
   "SafetyDoorInterface".fDoor9Interface.monitoring.DoorClose := #_w1 AND NOT "Safety.DataFromSafety".fDoorSwitchStatus.stk2NgBoxDoorOpen AND NOT "SafetyDoorInterface".fDoor9Interface.monitoring.DoorOpen;
   "SafetyDoorInterface".fDoor9Interface.monitoring.DoorLock := #_w1;
END_REGION

REGION Network 18: fDoor9 Command
   RUNG wire#powerrail
      Contact( #TRUE )
      wire#w1
      Contact( "SafetyDoorInterface".fDoor9Interface.commands.Lock )
      Coil( "Safety.DataToSafety".fDoor9Interface.Lock )
   END_RUNG
   RUNG wire#w1
      Contact( "SafetyDoorInterface".fDoor9Interface.commands.Unlock )
      Coil( "Safety.DataToSafety".fDoor9Interface.Unlock )
   END_RUNG
   // the same network as SCL:
   "Safety.DataToSafety".fDoor9Interface.Lock := #TRUE AND "SafetyDoorInterface".fDoor9Interface.commands.Lock;
   "Safety.DataToSafety".fDoor9Interface.Unlock := #TRUE AND "SafetyDoorInterface".fDoor9Interface.commands.Unlock;
END_REGION

REGION Network 19: fDoor10 monitoring
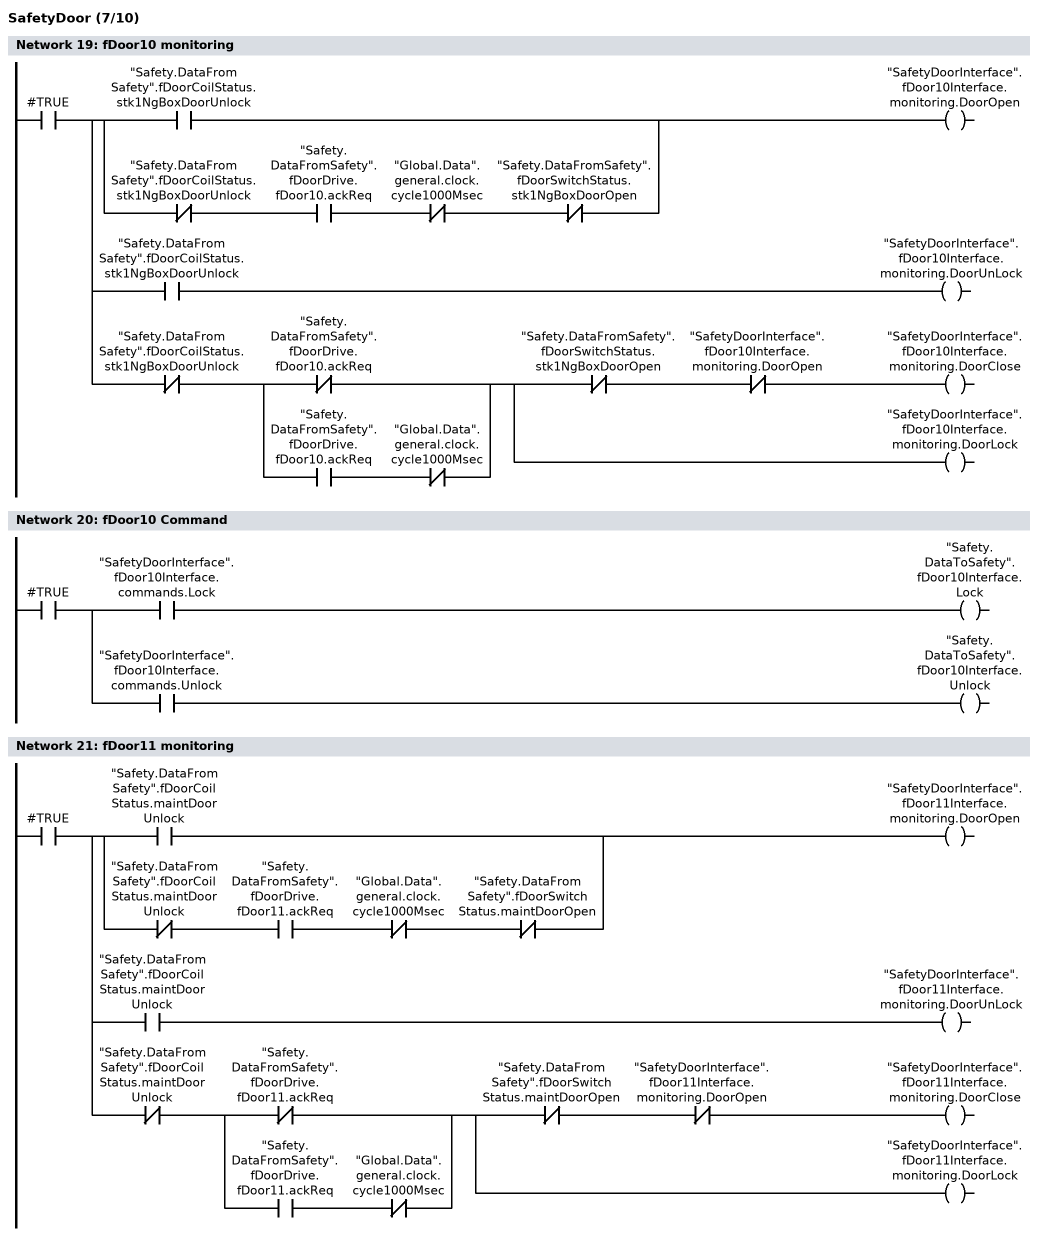
   RUNG wire#powerrail
      Contact( #TRUE )
      wire#w1
      Contact( "Safety.DataFromSafety".fDoorCoilStatus.stk1NgBoxDoorUnlock )
      wire#w2
      Coil( "SafetyDoorInterface".fDoor10Interface.monitoring.DoorOpen )
   END_RUNG
   RUNG wire#w1
      I_Contact( "Safety.DataFromSafety".fDoorCoilStatus.stk1NgBoxDoorUnlock )
      Contact( "Safety.DataFromSafety".fDoorDrive.fDoor10.ackReq )
      I_Contact( "Global.Data".general.clock.cycle1000Msec )
      I_Contact( "Safety.DataFromSafety".fDoorSwitchStatus.stk1NgBoxDoorOpen )
   END_RUNG wire#w2
   RUNG wire#w1
      Contact( "Safety.DataFromSafety".fDoorCoilStatus.stk1NgBoxDoorUnlock )
      Coil( "SafetyDoorInterface".fDoor10Interface.monitoring.DoorUnLock )
   END_RUNG
   RUNG wire#w1
      I_Contact( "Safety.DataFromSafety".fDoorCoilStatus.stk1NgBoxDoorUnlock )
      wire#w3
      I_Contact( "Safety.DataFromSafety".fDoorDrive.fDoor10.ackReq )
      wire#w4
      I_Contact( "Safety.DataFromSafety".fDoorSwitchStatus.stk1NgBoxDoorOpen )
      I_Contact( "SafetyDoorInterface".fDoor10Interface.monitoring.DoorOpen )
      Coil( "SafetyDoorInterface".fDoor10Interface.monitoring.DoorClose )
   END_RUNG
   RUNG wire#w3
      Contact( "Safety.DataFromSafety".fDoorDrive.fDoor10.ackReq )
      I_Contact( "Global.Data".general.clock.cycle1000Msec )
   END_RUNG wire#w4
   RUNG wire#w4
      Coil( "SafetyDoorInterface".fDoor10Interface.monitoring.DoorLock )
   END_RUNG
   // the same network as SCL:
   "SafetyDoorInterface".fDoor10Interface.monitoring.DoorOpen := #TRUE AND ("Safety.DataFromSafety".fDoorCoilStatus.stk1NgBoxDoorUnlock OR (NOT "Safety.DataFromSafety".fDoorCoilStatus.stk1NgBoxDoorUnlock AND "Safety.DataFromSafety".fDoorDrive.fDoor10.ackReq AND NOT "Global.Data".general.clock.cycle1000Msec AND NOT "Safety.DataFromSafety".fDoorSwitchStatus.stk1NgBoxDoorOpen));
   "SafetyDoorInterface".fDoor10Interface.monitoring.DoorUnLock := #TRUE AND "Safety.DataFromSafety".fDoorCoilStatus.stk1NgBoxDoorUnlock;
   #_w1 := #TRUE AND NOT "Safety.DataFromSafety".fDoorCoilStatus.stk1NgBoxDoorUnlock AND (NOT "Safety.DataFromSafety".fDoorDrive.fDoor10.ackReq OR ("Safety.DataFromSafety".fDoorDrive.fDoor10.ackReq AND NOT "Global.Data".general.clock.cycle1000Msec));
   "SafetyDoorInterface".fDoor10Interface.monitoring.DoorClose := #_w1 AND NOT "Safety.DataFromSafety".fDoorSwitchStatus.stk1NgBoxDoorOpen AND NOT "SafetyDoorInterface".fDoor10Interface.monitoring.DoorOpen;
   "SafetyDoorInterface".fDoor10Interface.monitoring.DoorLock := #_w1;
END_REGION

REGION Network 20: fDoor10 Command
   RUNG wire#powerrail
      Contact( #TRUE )
      wire#w1
      Contact( "SafetyDoorInterface".fDoor10Interface.commands.Lock )
      Coil( "Safety.DataToSafety".fDoor10Interface.Lock )
   END_RUNG
   RUNG wire#w1
      Contact( "SafetyDoorInterface".fDoor10Interface.commands.Unlock )
      Coil( "Safety.DataToSafety".fDoor10Interface.Unlock )
   END_RUNG
   // the same network as SCL:
   "Safety.DataToSafety".fDoor10Interface.Lock := #TRUE AND "SafetyDoorInterface".fDoor10Interface.commands.Lock;
   "Safety.DataToSafety".fDoor10Interface.Unlock := #TRUE AND "SafetyDoorInterface".fDoor10Interface.commands.Unlock;
END_REGION

REGION Network 21: fDoor11 monitoring
   RUNG wire#powerrail
      Contact( #TRUE )
      wire#w1
      Contact( "Safety.DataFromSafety".fDoorCoilStatus.maintDoorUnlock )
      wire#w2
      Coil( "SafetyDoorInterface".fDoor11Interface.monitoring.DoorOpen )
   END_RUNG
   RUNG wire#w1
      I_Contact( "Safety.DataFromSafety".fDoorCoilStatus.maintDoorUnlock )
      Contact( "Safety.DataFromSafety".fDoorDrive.fDoor11.ackReq )
      I_Contact( "Global.Data".general.clock.cycle1000Msec )
      I_Contact( "Safety.DataFromSafety".fDoorSwitchStatus.maintDoorOpen )
   END_RUNG wire#w2
   RUNG wire#w1
      Contact( "Safety.DataFromSafety".fDoorCoilStatus.maintDoorUnlock )
      Coil( "SafetyDoorInterface".fDoor11Interface.monitoring.DoorUnLock )
   END_RUNG
   RUNG wire#w1
      I_Contact( "Safety.DataFromSafety".fDoorCoilStatus.maintDoorUnlock )
      wire#w3
      I_Contact( "Safety.DataFromSafety".fDoorDrive.fDoor11.ackReq )
      wire#w4
      I_Contact( "Safety.DataFromSafety".fDoorSwitchStatus.maintDoorOpen )
      I_Contact( "SafetyDoorInterface".fDoor11Interface.monitoring.DoorOpen )
      Coil( "SafetyDoorInterface".fDoor11Interface.monitoring.DoorClose )
   END_RUNG
   RUNG wire#w3
      Contact( "Safety.DataFromSafety".fDoorDrive.fDoor11.ackReq )
      I_Contact( "Global.Data".general.clock.cycle1000Msec )
   END_RUNG wire#w4
   RUNG wire#w4
      Coil( "SafetyDoorInterface".fDoor11Interface.monitoring.DoorLock )
   END_RUNG
   // the same network as SCL:
   "SafetyDoorInterface".fDoor11Interface.monitoring.DoorOpen := #TRUE AND ("Safety.DataFromSafety".fDoorCoilStatus.maintDoorUnlock OR (NOT "Safety.DataFromSafety".fDoorCoilStatus.maintDoorUnlock AND "Safety.DataFromSafety".fDoorDrive.fDoor11.ackReq AND NOT "Global.Data".general.clock.cycle1000Msec AND NOT "Safety.DataFromSafety".fDoorSwitchStatus.maintDoorOpen));
   "SafetyDoorInterface".fDoor11Interface.monitoring.DoorUnLock := #TRUE AND "Safety.DataFromSafety".fDoorCoilStatus.maintDoorUnlock;
   #_w1 := #TRUE AND NOT "Safety.DataFromSafety".fDoorCoilStatus.maintDoorUnlock AND (NOT "Safety.DataFromSafety".fDoorDrive.fDoor11.ackReq OR ("Safety.DataFromSafety".fDoorDrive.fDoor11.ackReq AND NOT "Global.Data".general.clock.cycle1000Msec));
   "SafetyDoorInterface".fDoor11Interface.monitoring.DoorClose := #_w1 AND NOT "Safety.DataFromSafety".fDoorSwitchStatus.maintDoorOpen AND NOT "SafetyDoorInterface".fDoor11Interface.monitoring.DoorOpen;
   "SafetyDoorInterface".fDoor11Interface.monitoring.DoorLock := #_w1;
END_REGION

REGION Network 22: fDoor11 Command
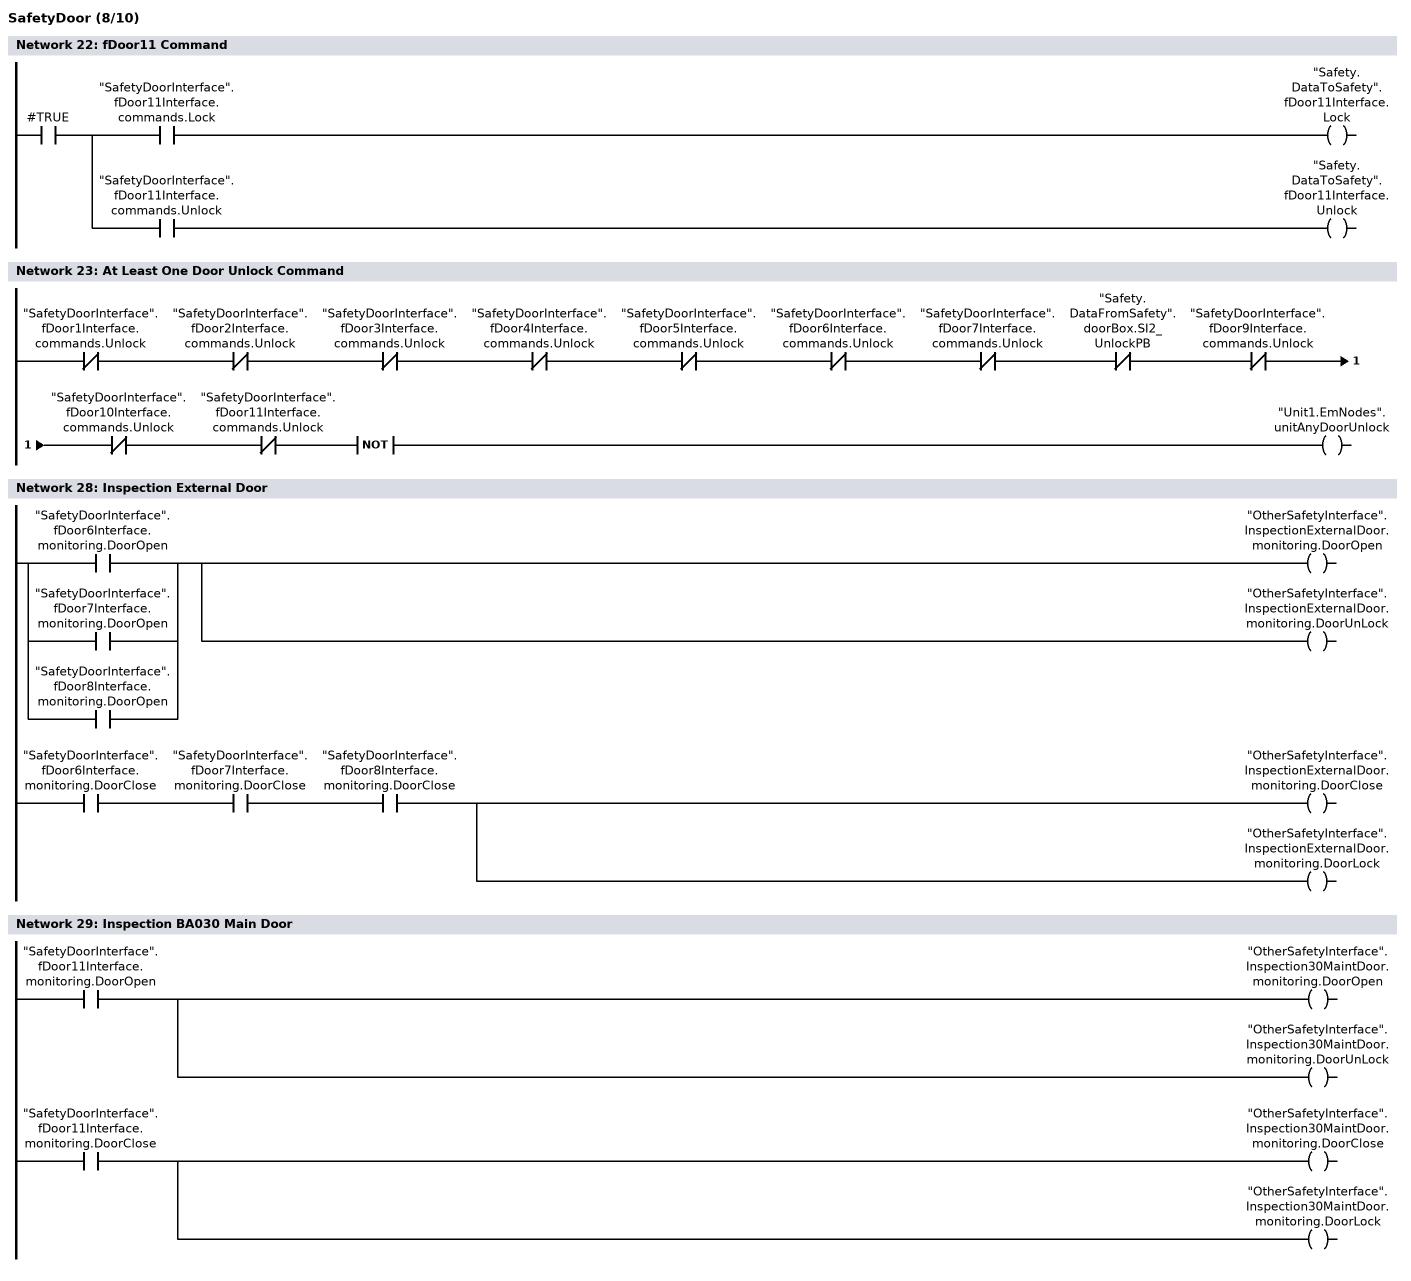
   RUNG wire#powerrail
      Contact( #TRUE )
      wire#w1
      Contact( "SafetyDoorInterface".fDoor11Interface.commands.Lock )
      Coil( "Safety.DataToSafety".fDoor11Interface.Lock )
   END_RUNG
   RUNG wire#w1
      Contact( "SafetyDoorInterface".fDoor11Interface.commands.Unlock )
      Coil( "Safety.DataToSafety".fDoor11Interface.Unlock )
   END_RUNG
   // the same network as SCL:
   "Safety.DataToSafety".fDoor11Interface.Lock := #TRUE AND "SafetyDoorInterface".fDoor11Interface.commands.Lock;
   "Safety.DataToSafety".fDoor11Interface.Unlock := #TRUE AND "SafetyDoorInterface".fDoor11Interface.commands.Unlock;
END_REGION

REGION Network 23: At Least One Door Unlock Command
   RUNG wire#powerrail
      I_Contact( "SafetyDoorInterface".fDoor1Interface.commands.Unlock )
      I_Contact( "SafetyDoorInterface".fDoor2Interface.commands.Unlock )
      I_Contact( "SafetyDoorInterface".fDoor3Interface.commands.Unlock )
      I_Contact( "SafetyDoorInterface".fDoor4Interface.commands.Unlock )
      I_Contact( "SafetyDoorInterface".fDoor5Interface.commands.Unlock )
      I_Contact( "SafetyDoorInterface".fDoor6Interface.commands.Unlock )
      I_Contact( "SafetyDoorInterface".fDoor7Interface.commands.Unlock )
      I_Contact( "Safety.DataFromSafety".doorBox.SI2_UnlockPB )
      I_Contact( "SafetyDoorInterface".fDoor9Interface.commands.Unlock )
      I_Contact( "SafetyDoorInterface".fDoor10Interface.commands.Unlock )
      I_Contact( "SafetyDoorInterface".fDoor11Interface.commands.Unlock )
      Not()
      Coil( "Unit1.EmNodes".unitAnyDoorUnlock )
   END_RUNG
   // the same network as SCL:
   "Unit1.EmNodes".unitAnyDoorUnlock := NOT (NOT "SafetyDoorInterface".fDoor1Interface.commands.Unlock AND NOT "SafetyDoorInterface".fDoor2Interface.commands.Unlock AND NOT "SafetyDoorInterface".fDoor3Interface.commands.Unlock AND NOT "SafetyDoorInterface".fDoor4Interface.commands.Unlock AND NOT "SafetyDoorInterface".fDoor5Interface.commands.Unlock AND NOT "SafetyDoorInterface".fDoor6Interface.commands.Unlock AND NOT "SafetyDoorInterface".fDoor7Interface.commands.Unlock AND NOT "Safety.DataFromSafety".doorBox.SI2_UnlockPB AND NOT "SafetyDoorInterface".fDoor9Interface.commands.Unlock AND NOT "SafetyDoorInterface".fDoor10Interface.commands.Unlock AND NOT "SafetyDoorInterface".fDoor11Interface.commands.Unlock);
END_REGION

REGION Network 24: BA010 Other Door
END_REGION

REGION Network 25: BA015 Other Door
END_REGION

REGION Network 26: BA030 Other Door
END_REGION

REGION Network 27: BA040 Other Door
END_REGION

REGION Network 28: Inspection External Door
   RUNG wire#powerrail
      Contact( "SafetyDoorInterface".fDoor6Interface.monitoring.DoorOpen )
      wire#w1
      Coil( "OtherSafetyInterface".InspectionExternalDoor.monitoring.DoorOpen )
   END_RUNG
   RUNG wire#powerrail
      Contact( "SafetyDoorInterface".fDoor7Interface.monitoring.DoorOpen )
   END_RUNG wire#w1
   RUNG wire#powerrail
      Contact( "SafetyDoorInterface".fDoor8Interface.monitoring.DoorOpen )
   END_RUNG wire#w1
   RUNG wire#w1
      Coil( "OtherSafetyInterface".InspectionExternalDoor.monitoring.DoorUnLock )
   END_RUNG
   RUNG wire#powerrail
      Contact( "SafetyDoorInterface".fDoor6Interface.monitoring.DoorClose )
      Contact( "SafetyDoorInterface".fDoor7Interface.monitoring.DoorClose )
      Contact( "SafetyDoorInterface".fDoor8Interface.monitoring.DoorClose )
      wire#w2
      Coil( "OtherSafetyInterface".InspectionExternalDoor.monitoring.DoorClose )
   END_RUNG
   RUNG wire#w2
      Coil( "OtherSafetyInterface".InspectionExternalDoor.monitoring.DoorLock )
   END_RUNG
   // the same network as SCL:
   "OtherSafetyInterface".InspectionExternalDoor.monitoring.DoorOpen := "SafetyDoorInterface".fDoor6Interface.monitoring.DoorOpen OR "SafetyDoorInterface".fDoor7Interface.monitoring.DoorOpen OR "SafetyDoorInterface".fDoor8Interface.monitoring.DoorOpen;
   "OtherSafetyInterface".InspectionExternalDoor.monitoring.DoorUnLock := "OtherSafetyInterface".InspectionExternalDoor.monitoring.DoorOpen;
   "OtherSafetyInterface".InspectionExternalDoor.monitoring.DoorClose := "SafetyDoorInterface".fDoor6Interface.monitoring.DoorClose AND "SafetyDoorInterface".fDoor7Interface.monitoring.DoorClose AND "SafetyDoorInterface".fDoor8Interface.monitoring.DoorClose;
   "OtherSafetyInterface".InspectionExternalDoor.monitoring.DoorLock := "OtherSafetyInterface".InspectionExternalDoor.monitoring.DoorClose;
END_REGION

REGION Network 29: Inspection BA030 Main Door
   RUNG wire#powerrail
      Contact( "SafetyDoorInterface".fDoor11Interface.monitoring.DoorOpen )
      wire#w1
      Coil( "OtherSafetyInterface".Inspection30MaintDoor.monitoring.DoorOpen )
   END_RUNG
   RUNG wire#w1
      Coil( "OtherSafetyInterface".Inspection30MaintDoor.monitoring.DoorUnLock )
   END_RUNG
   RUNG wire#powerrail
      Contact( "SafetyDoorInterface".fDoor11Interface.monitoring.DoorClose )
      wire#w2
      Coil( "OtherSafetyInterface".Inspection30MaintDoor.monitoring.DoorClose )
   END_RUNG
   RUNG wire#w2
      Coil( "OtherSafetyInterface".Inspection30MaintDoor.monitoring.DoorLock )
   END_RUNG
   // the same network as SCL:
   "OtherSafetyInterface".Inspection30MaintDoor.monitoring.DoorOpen := "SafetyDoorInterface".fDoor11Interface.monitoring.DoorOpen;
   "OtherSafetyInterface".Inspection30MaintDoor.monitoring.DoorUnLock := "SafetyDoorInterface".fDoor11Interface.monitoring.DoorOpen;
   "OtherSafetyInterface".Inspection30MaintDoor.monitoring.DoorClose := "SafetyDoorInterface".fDoor11Interface.monitoring.DoorClose;
   "OtherSafetyInterface".Inspection30MaintDoor.monitoring.DoorLock := "SafetyDoorInterface".fDoor11Interface.monitoring.DoorClose;
END_REGION

REGION Network 30: Inspection BA040 Main Door
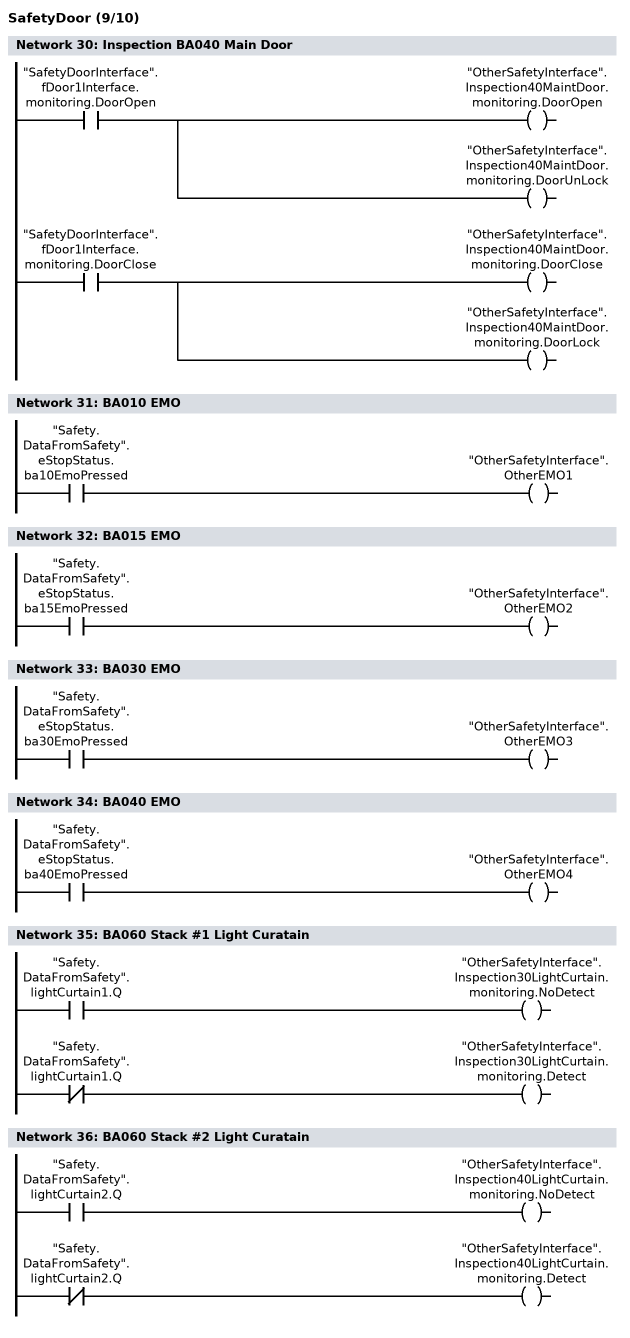
   RUNG wire#powerrail
      Contact( "SafetyDoorInterface".fDoor1Interface.monitoring.DoorOpen )
      wire#w1
      Coil( "OtherSafetyInterface".Inspection40MaintDoor.monitoring.DoorOpen )
   END_RUNG
   RUNG wire#w1
      Coil( "OtherSafetyInterface".Inspection40MaintDoor.monitoring.DoorUnLock )
   END_RUNG
   RUNG wire#powerrail
      Contact( "SafetyDoorInterface".fDoor1Interface.monitoring.DoorClose )
      wire#w2
      Coil( "OtherSafetyInterface".Inspection40MaintDoor.monitoring.DoorClose )
   END_RUNG
   RUNG wire#w2
      Coil( "OtherSafetyInterface".Inspection40MaintDoor.monitoring.DoorLock )
   END_RUNG
   // the same network as SCL:
   "OtherSafetyInterface".Inspection40MaintDoor.monitoring.DoorOpen := "SafetyDoorInterface".fDoor1Interface.monitoring.DoorOpen;
   "OtherSafetyInterface".Inspection40MaintDoor.monitoring.DoorUnLock := "SafetyDoorInterface".fDoor1Interface.monitoring.DoorOpen;
   "OtherSafetyInterface".Inspection40MaintDoor.monitoring.DoorClose := "SafetyDoorInterface".fDoor1Interface.monitoring.DoorClose;
   "OtherSafetyInterface".Inspection40MaintDoor.monitoring.DoorLock := "SafetyDoorInterface".fDoor1Interface.monitoring.DoorClose;
END_REGION

REGION Network 31: BA010 EMO
   RUNG wire#powerrail
      Contact( "Safety.DataFromSafety".eStopStatus.ba10EmoPressed )
      Coil( "OtherSafetyInterface".OtherEMO1 )
   END_RUNG
   // the same network as SCL:
   "OtherSafetyInterface".OtherEMO1 := "Safety.DataFromSafety".eStopStatus.ba10EmoPressed;
END_REGION

REGION Network 32: BA015 EMO
   RUNG wire#powerrail
      Contact( "Safety.DataFromSafety".eStopStatus.ba15EmoPressed )
      Coil( "OtherSafetyInterface".OtherEMO2 )
   END_RUNG
   // the same network as SCL:
   "OtherSafetyInterface".OtherEMO2 := "Safety.DataFromSafety".eStopStatus.ba15EmoPressed;
END_REGION

REGION Network 33: BA030 EMO
   RUNG wire#powerrail
      Contact( "Safety.DataFromSafety".eStopStatus.ba30EmoPressed )
      Coil( "OtherSafetyInterface".OtherEMO3 )
   END_RUNG
   // the same network as SCL:
   "OtherSafetyInterface".OtherEMO3 := "Safety.DataFromSafety".eStopStatus.ba30EmoPressed;
END_REGION

REGION Network 34: BA040 EMO
   RUNG wire#powerrail
      Contact( "Safety.DataFromSafety".eStopStatus.ba40EmoPressed )
      Coil( "OtherSafetyInterface".OtherEMO4 )
   END_RUNG
   // the same network as SCL:
   "OtherSafetyInterface".OtherEMO4 := "Safety.DataFromSafety".eStopStatus.ba40EmoPressed;
END_REGION

REGION Network 35: BA060 Stack #1 Light Curatain
   RUNG wire#powerrail
      Contact( "Safety.DataFromSafety".lightCurtain1.Q )
      Coil( "OtherSafetyInterface".Inspection30LightCurtain.monitoring.NoDetect )
   END_RUNG
   RUNG wire#powerrail
      I_Contact( "Safety.DataFromSafety".lightCurtain1.Q )
      Coil( "OtherSafetyInterface".Inspection30LightCurtain.monitoring.Detect )
   END_RUNG
   // the same network as SCL:
   "OtherSafetyInterface".Inspection30LightCurtain.monitoring.NoDetect := "Safety.DataFromSafety".lightCurtain1.Q;
   "OtherSafetyInterface".Inspection30LightCurtain.monitoring.Detect := NOT "Safety.DataFromSafety".lightCurtain1.Q;
END_REGION

REGION Network 36: BA060 Stack #2 Light Curatain
   RUNG wire#powerrail
      Contact( "Safety.DataFromSafety".lightCurtain2.Q )
      Coil( "OtherSafetyInterface".Inspection40LightCurtain.monitoring.NoDetect )
   END_RUNG
   RUNG wire#powerrail
      I_Contact( "Safety.DataFromSafety".lightCurtain2.Q )
      Coil( "OtherSafetyInterface".Inspection40LightCurtain.monitoring.Detect )
   END_RUNG
   // the same network as SCL:
   "OtherSafetyInterface".Inspection40LightCurtain.monitoring.NoDetect := "Safety.DataFromSafety".lightCurtain2.Q;
   "OtherSafetyInterface".Inspection40LightCurtain.monitoring.Detect := NOT "Safety.DataFromSafety".lightCurtain2.Q;
END_REGION

REGION Network 37: BA030 Cathode Conveyor Cover
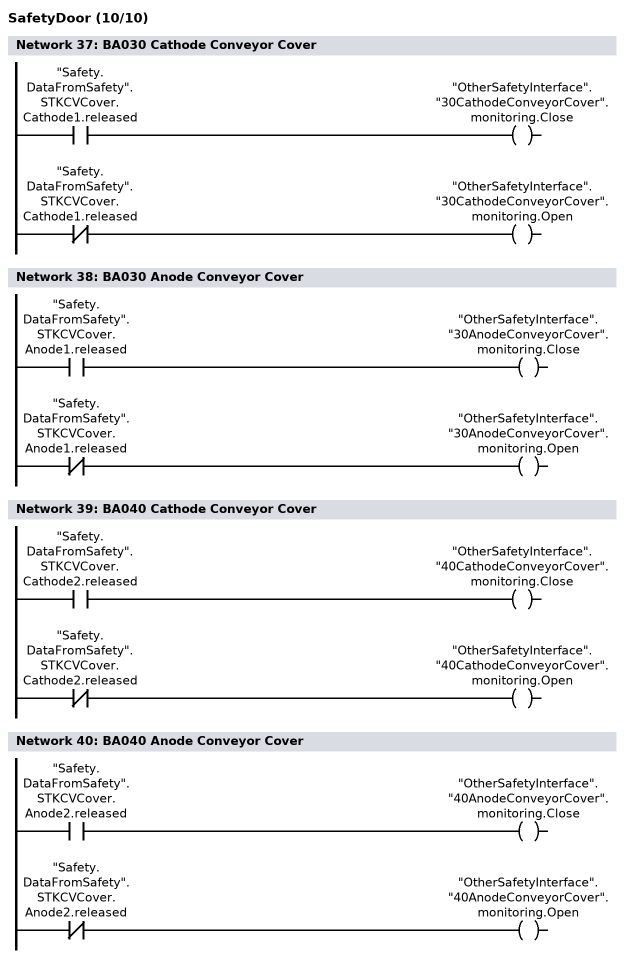
   RUNG wire#powerrail
      Contact( "Safety.DataFromSafety".STKCVCover.Cathode1.released )
      Coil( "OtherSafetyInterface"."30CathodeConveyorCover".monitoring.Close )
   END_RUNG
   RUNG wire#powerrail
      I_Contact( "Safety.DataFromSafety".STKCVCover.Cathode1.released )
      Coil( "OtherSafetyInterface"."30CathodeConveyorCover".monitoring.Open )
   END_RUNG
   // the same network as SCL:
   "OtherSafetyInterface"."30CathodeConveyorCover".monitoring.Close := "Safety.DataFromSafety".STKCVCover.Cathode1.released;
   "OtherSafetyInterface"."30CathodeConveyorCover".monitoring.Open := NOT "Safety.DataFromSafety".STKCVCover.Cathode1.released;
END_REGION

REGION Network 38: BA030 Anode Conveyor Cover
   RUNG wire#powerrail
      Contact( "Safety.DataFromSafety".STKCVCover.Anode1.released )
      Coil( "OtherSafetyInterface"."30AnodeConveyorCover".monitoring.Close )
   END_RUNG
   RUNG wire#powerrail
      I_Contact( "Safety.DataFromSafety".STKCVCover.Anode1.released )
      Coil( "OtherSafetyInterface"."30AnodeConveyorCover".monitoring.Open )
   END_RUNG
   // the same network as SCL:
   "OtherSafetyInterface"."30AnodeConveyorCover".monitoring.Close := "Safety.DataFromSafety".STKCVCover.Anode1.released;
   "OtherSafetyInterface"."30AnodeConveyorCover".monitoring.Open := NOT "Safety.DataFromSafety".STKCVCover.Anode1.released;
END_REGION

REGION Network 39: BA040 Cathode Conveyor Cover
   RUNG wire#powerrail
      Contact( "Safety.DataFromSafety".STKCVCover.Cathode2.released )
      Coil( "OtherSafetyInterface"."40CathodeConveyorCover".monitoring.Close )
   END_RUNG
   RUNG wire#powerrail
      I_Contact( "Safety.DataFromSafety".STKCVCover.Cathode2.released )
      Coil( "OtherSafetyInterface"."40CathodeConveyorCover".monitoring.Open )
   END_RUNG
   // the same network as SCL:
   "OtherSafetyInterface"."40CathodeConveyorCover".monitoring.Close := "Safety.DataFromSafety".STKCVCover.Cathode2.released;
   "OtherSafetyInterface"."40CathodeConveyorCover".monitoring.Open := NOT "Safety.DataFromSafety".STKCVCover.Cathode2.released;
END_REGION

REGION Network 40: BA040 Anode Conveyor Cover
   RUNG wire#powerrail
      Contact( "Safety.DataFromSafety".STKCVCover.Anode2.released )
      Coil( "OtherSafetyInterface"."40AnodeConveyorCover".monitoring.Close )
   END_RUNG
   RUNG wire#powerrail
      I_Contact( "Safety.DataFromSafety".STKCVCover.Anode2.released )
      Coil( "OtherSafetyInterface"."40AnodeConveyorCover".monitoring.Open )
   END_RUNG
   // the same network as SCL:
   "OtherSafetyInterface"."40AnodeConveyorCover".monitoring.Close := "Safety.DataFromSafety".STKCVCover.Anode2.released;
   "OtherSafetyInterface"."40AnodeConveyorCover".monitoring.Open := NOT "Safety.DataFromSafety".STKCVCover.Anode2.released;
END_REGION
END_FUNCTION
